PROGRAM MAIN
VAR

END_VAR

// System Control
PLCSystem.iTaskIdx  := GETCURTASKINDEXEX();
System(iTaskIdx 	:= PLCSystem.iTaskIdx,
	   bFirstCycle  := PLCSystem.bFirstCycle);

ServoGVLs.coeRead(Axis:= servoGVLs.servo1Interface.ioAxisRef,
				  Index := 16#2191,
				  SubIndex := 16#01,
				  Execute := servoGVLs.toggle,
				  Busy =>,
				  pDstBuf := ADR(servoGVLs.catchWord),
				  BufLen := SIZEOF(servoGVLs.catchWord));

// TCP Connection

TCPComm(cmdData => gvlMotion.cmdData);
// Mode Control
gvlMotion.autoMode := NOT gvlMotion.manualMode;
IF gvlMotion.manualMode THEN
	gvlMotion.servo1(stServoInterface := servoGVLs.servo1Interface);
END_IF
// Servo 1 Auto Control via Server
gvlMotion.bank1(
	   cmdData := gvlMotion.cmdData,
	   bEnableDrive := gvlMotion.bEnableDrive,
	   bStartDrive := gvlMotion.bStartDrive,
	   bInterlockOK := gvlMotion.bInterlockOK,
	   bTriggerDefault := gvlMotion.bTriggerDefault,
	   driveStatus => gvlMotion.driveStatus,
	   mcBankAxis := ServoGVLs.servo1Interface);

END_PROGRAM

(* stored: Version 1.1.0.1, ProductVersion 3.1.4024.12
   POU MAIN: Id {9767283b-cca1-4624-be02-ae2381d3ffbe}, SpecialFunc None *)
